// TIA Portal V18 export
FUNCTION "FC_Write_Actual_Recipe_To_Devices" : Void   // FC5, SCL
{ S7_Optimized_Access := 'TRUE' }
// =============================================================================
//  AUTHOR      : Gemini
//  FAMILY      : Recipe
//  NAME        : LoadToDev
//  DESCRIPTION : Writes ACTUAL_CHOOSEN_TYPE parameters to Device DBs and Logic Buffers
//                Exact reverse operation of FC_Save_Values_Final
// =============================================================================
// stored: SetENOAutomatically false
   VAR_TEMP
      i : Int;
   END_VAR
BEGIN


     //=============================================================================
     // use recipe trigger
     //=============================================================================


   IF "DB_PARAMETERS_TEACH".HMI_PAGE_CONTROL.Use_recipe_trigger AND "DB_PARAMETERS_TEACH".HMI_PAGE_CONTROL.Use_recipe_Nbr <> 0
   THEN



     "DB_ALL_PROCESS_PARAMETERS".ACTUAL_CHOOSEN_TYPE := "DB_ALL_PROCESS_PARAMETERS".PRODUCT_TYPE["DB_PARAMETERS_TEACH".HMI_PAGE_CONTROL.Use_recipe_Nbr];
     //=============================================================================
     // 1. MOTION - IAI AXES (Write to IAI_Ax.Auto.Pos[...])
     //=============================================================================
     FOR #i := 1 TO 20 DO
       // IAI_A1 (Gluing Nozzle Z)
       "IAI_A1".Auto.Pos[#i].Pos :=
       "DB_ALL_PROCESS_PARAMETERS".ACTUAL_CHOOSEN_TYPE.Motion.Gluing_Nozzle_Z.Position[#i].Pos;
       "IAI_A1".Auto.Pos[#i].Vel :=
       "DB_ALL_PROCESS_PARAMETERS".ACTUAL_CHOOSEN_TYPE.Motion.Gluing_Nozzle_Z.Position[#i].Vel;

       // IAI_A2 (Gluing Nozzle X)
       "IAI_A2".Auto.Pos[#i].Pos :=
       "DB_ALL_PROCESS_PARAMETERS".ACTUAL_CHOOSEN_TYPE.Motion.Gluing_Nozzle_X.Position[#i].Pos;
       "IAI_A2".Auto.Pos[#i].Vel :=
       "DB_ALL_PROCESS_PARAMETERS".ACTUAL_CHOOSEN_TYPE.Motion.Gluing_Nozzle_X.Position[#i].Vel;

       // IAI_A3 (Gluing Nozzle Y)
       "IAI_A3".Auto.Pos[#i].Pos :=
       "DB_ALL_PROCESS_PARAMETERS".ACTUAL_CHOOSEN_TYPE.Motion.Gluing_Nozzle_Y.Position[#i].Pos;
       "IAI_A3".Auto.Pos[#i].Vel :=
       "DB_ALL_PROCESS_PARAMETERS".ACTUAL_CHOOSEN_TYPE.Motion.Gluing_Nozzle_Y.Position[#i].Vel;
     END_FOR;

     //=============================================================================
     // 2. MOTION - V90 AXES (Write to ServoV90_Ax.Auto.Pos[...])
     //=============================================================================
     FOR #i := 1 TO 20 DO
       // ServoV90_A1 (Ring Turntable Axis 1)
       "ServoV90_A1".Auto.Pos[#i].Pos :=
       "DB_ALL_PROCESS_PARAMETERS".ACTUAL_CHOOSEN_TYPE.Motion.Ring_Turntable_Axis_1.Position[#i].Pos;
       "ServoV90_A1".Auto.Pos[#i].Vel :=
       "DB_ALL_PROCESS_PARAMETERS".ACTUAL_CHOOSEN_TYPE.Motion.Ring_Turntable_Axis_1.Position[#i].Vel;

       // ServoV90_A2 (Shaft Scan Turntable)
       "ServoV90_A2".Auto.Pos[#i].Pos :=
       "DB_ALL_PROCESS_PARAMETERS".ACTUAL_CHOOSEN_TYPE.Motion.Shaft_Scan_Turntable_Axis.Position[#i].Pos;
       "ServoV90_A2".Auto.Pos[#i].Vel :=
       "DB_ALL_PROCESS_PARAMETERS".ACTUAL_CHOOSEN_TYPE.Motion.Shaft_Scan_Turntable_Axis.Position[#i].Vel;

       // ServoV90_A3 (Gluing Rotary Jig)
       "ServoV90_A3".Auto.Pos[#i].Pos :=
       "DB_ALL_PROCESS_PARAMETERS".ACTUAL_CHOOSEN_TYPE.Motion.Gluing_Rotary_Jig_Axis.Position[#i].Pos;
       "ServoV90_A3".Auto.Pos[#i].Vel :=
       "DB_ALL_PROCESS_PARAMETERS".ACTUAL_CHOOSEN_TYPE.Motion.Gluing_Rotary_Jig_Axis.Position[#i].Vel;

       // ServoV90_A4 (Ring Turntable 2)
       "ServoV90_A4".Auto.Pos[#i].Pos :=
       "DB_ALL_PROCESS_PARAMETERS".ACTUAL_CHOOSEN_TYPE.Motion.Ring_Turntable_Axis_2.Position[#i].Pos;
       "ServoV90_A4".Auto.Pos[#i].Vel :=
       "DB_ALL_PROCESS_PARAMETERS".ACTUAL_CHOOSEN_TYPE.Motion.Ring_Turntable_Axis_2.Position[#i].Vel;
     END_FOR;

     //=============================================================================
     // 3. PARAMETER ELEMENTS (Write to ST10_RecipeDB - Logic Buffer)
     //=============================================================================

     // --- Press Programs ---
     "ST10_RecipeDB".ParameterElement.B1PressProgram := "DB_ALL_PROCESS_PARAMETERS".ACTUAL_CHOOSEN_TYPE.Process.Press.B1_Program;
     "ST10_RecipeDB".ParameterElement.B2PressProgram := "DB_ALL_PROCESS_PARAMETERS".ACTUAL_CHOOSEN_TYPE.Process.Press.B2_Program;

     // --- Vision Programs (IV3) ---
     "ST10_RecipeDB".ParameterElement.CGlueShaftIV3Program_1 := "DB_ALL_PROCESS_PARAMETERS".ACTUAL_CHOOSEN_TYPE.Process.Vision.CGlueShaftIV3_Progs[1];
     "ST10_RecipeDB".ParameterElement.CGlueShaftIV3Program_2 := "DB_ALL_PROCESS_PARAMETERS".ACTUAL_CHOOSEN_TYPE.Process.Vision.CGlueShaftIV3_Progs[2];
     "ST10_RecipeDB".ParameterElement.CGlueShaftIV3Program_3 := "DB_ALL_PROCESS_PARAMETERS".ACTUAL_CHOOSEN_TYPE.Process.Vision.CGlueShaftIV3_Progs[3];
     "ST10_RecipeDB".ParameterElement.CGlueShaftIV3Program_4 := "DB_ALL_PROCESS_PARAMETERS".ACTUAL_CHOOSEN_TYPE.Process.Vision.CGlueShaftIV3_Progs[4];

     "ST10_RecipeDB".ParameterElement.CGlueMagnetIV3Program := "DB_ALL_PROCESS_PARAMETERS".ACTUAL_CHOOSEN_TYPE.Process.Vision.CGlueMagnetIV3_Prog;
     "ST10_RecipeDB".ParameterElement.CGlueProgram := "DB_ALL_PROCESS_PARAMETERS".ACTUAL_CHOOSEN_TYPE.Process.Vision.CGlueProgram;

     // --- Tooling Codes (Robot 1) ---
     "ST10_RecipeDB".ParameterElement.R1GripperFixtureCode[1] := "DB_ALL_PROCESS_PARAMETERS".ACTUAL_CHOOSEN_TYPE."Tooling Code".ROB1_Shaft_Handling_Robot.Gripper."JAW TOOLING LEFT";
     "ST10_RecipeDB".ParameterElement.R1GripperFixtureCode[2] := "DB_ALL_PROCESS_PARAMETERS".ACTUAL_CHOOSEN_TYPE."Tooling Code".ROB1_Shaft_Handling_Robot.Gripper."JAW TOOLING RIGHT";
     "ST10_RecipeDB".ParameterElement.R1GripperFixtureCode[3] := "DB_ALL_PROCESS_PARAMETERS".ACTUAL_CHOOSEN_TYPE."Tooling Code".ROB1_Shaft_Handling_Robot.Gripper."SHAFT CLAMPING LEFT";
     "ST10_RecipeDB".ParameterElement.R1GripperFixtureCode[4] := "DB_ALL_PROCESS_PARAMETERS".ACTUAL_CHOOSEN_TYPE."Tooling Code".ROB1_Shaft_Handling_Robot.Gripper."SHAFT CLAMPING RIGHT";

     // --- Tooling Codes (Robot 2) ---
     "ST10_RecipeDB".ParameterElement.R2GripperFixtureCode[1] := "DB_ALL_PROCESS_PARAMETERS".ACTUAL_CHOOSEN_TYPE."Tooling Code".ROB2_Main_Assembly_Robot.Gripper."JAW TOOLING LEFT";
     "ST10_RecipeDB".ParameterElement.R2GripperFixtureCode[2] := "DB_ALL_PROCESS_PARAMETERS".ACTUAL_CHOOSEN_TYPE."Tooling Code".ROB2_Main_Assembly_Robot.Gripper."JAW TOOLING RIGHT";
     "ST10_RecipeDB".ParameterElement.R2GripperFixtureCode[3] := "DB_ALL_PROCESS_PARAMETERS".ACTUAL_CHOOSEN_TYPE."Tooling Code".ROB2_Main_Assembly_Robot.Gripper."SHAFT CLAMPING LEFT";
     "ST10_RecipeDB".ParameterElement.R2GripperFixtureCode[4] := "DB_ALL_PROCESS_PARAMETERS".ACTUAL_CHOOSEN_TYPE."Tooling Code".ROB2_Main_Assembly_Robot.Gripper."SHAFT CLAMPING RIGHT";

     // --- Tooling Codes (Robot 3) ---
     "ST10_RecipeDB".ParameterElement.R3GripperFixtureCode[1] := "DB_ALL_PROCESS_PARAMETERS".ACTUAL_CHOOSEN_TYPE."Tooling Code".ROB3_Unloading_Robot.Gripper."JAW TOOLING LEFT";
     "ST10_RecipeDB".ParameterElement.R3GripperFixtureCode[2] := "DB_ALL_PROCESS_PARAMETERS".ACTUAL_CHOOSEN_TYPE."Tooling Code".ROB3_Unloading_Robot.Gripper."JAW TOOLING RIGHT";
     "ST10_RecipeDB".ParameterElement.R3GripperFixtureCode[3] := "DB_ALL_PROCESS_PARAMETERS".ACTUAL_CHOOSEN_TYPE."Tooling Code".ROB3_Unloading_Robot.Gripper."SHAFT CLAMPING LEFT";
     "ST10_RecipeDB".ParameterElement.R3GripperFixtureCode[4] := "DB_ALL_PROCESS_PARAMETERS".ACTUAL_CHOOSEN_TYPE."Tooling Code".ROB3_Unloading_Robot.Gripper."SHAFT CLAMPING RIGHT";

     // --- Table Fixture Codes (A1 & A2) ---
     // Using LOOP because Save function saves array elements individually or implicitly, but Load needs to fill the buffer
     FOR #i := 1 TO 8 DO
       "ST10_RecipeDB".ParameterElement.A1_TableFixtureCode[#i] := "DB_ALL_PROCESS_PARAMETERS".ACTUAL_CHOOSEN_TYPE."Tooling Code".A1_Table[#i];
       "ST10_RecipeDB".ParameterElement.A2_TableFixtureCode[#i] := "DB_ALL_PROCESS_PARAMETERS".ACTUAL_CHOOSEN_TYPE."Tooling Code".A2_Table[#i];
     END_FOR;

     "DB_PARAMETERS_TEACH".HMI_PAGE_CONTROL.Use_recipe_trigger := false;

   END_IF;
END_FUNCTION
